// TIA Portal V18 export
// export: Created 2026-06-12T02:00:00Z, ExportSetting WithDefaults
VAR_GLOBAL   // PLC tag table "PLC_AI_B3_Tags"
   AI_B3_Sequence_Count AT %MD0 : Real;   // COUNT 0-100
   AI_B3_Flow_CIP_Center AT %MD4 : Real;   // FLOW 100-200 L/h
   AI_B3_Temp_CIP_Upper AT %MD8 : Real;   // TEMP 50-80 °C
   AI_B3_Pressure_CIP_1 AT %MD12 : Real;   // PRESSURE 7-8 bar
   AI_B3_Temp_Chaff_1 AT %MD16 : Real;   // TEMP 50-80 °C
   AI_B3_Flow_CIP_Feed AT %MD20 : Real;   // FLOW 100-200 L/h
   AI_B3_Temp_Steam_1 AT %MD24 : Real;   // TEMP 50-80 °C
   AI_B3_Flow_UCWW_1 AT %MD28 : Real;   // FLOW 100-200 L/h
   AI_B3_RPM_Screw_Conv AT %MD32 : Real;   // RPM 800-1200 RPM
   AI_B3_Temp_Condensate_1 AT %MD36 : Real;   // TEMP 50-80 °C
   AI_B3_Pressure_Screw_1 AT %MD40 : Real;   // PRESSURE 7-8 bar
   AI_B3_Flow_CWW_Out AT %MD44 : Real;   // FLOW 100-200 L/h
   AI_B3_Pressure_CWW_1 AT %MD48 : Real;   // PRESSURE 7-8 bar
   AI_B3_Temp_Decanter2 AT %MD52 : Real;   // TEMP 50-80 °C
   AI_B3_RPM_Rotary2 AT %MD56 : Real;   // RPM 800-1200 RPM
   AI_B3_RPM_Rotary1 AT %MD60 : Real;   // RPM 800-1200 RPM
   AI_B3_Temp_GroundSilo AT %MD64 : Real;   // TEMP 50-80 °C
   AI_B3_Flow_GroundSilo AT %MD68 : Real;   // FLOW 100-200 L/h
   AI_B3_Pressure_Mid_1 AT %MD72 : Real;   // PRESSURE 7-8 bar
   AI_B3_Flow_Condensate AT %MD76 : Real;   // FLOW 100-200 L/h
   AI_B3_Flow_Sump_Out AT %MD80 : Real;   // FLOW 100-200 L/h
   AI_B3_Level_Sump AT %MD84 : Real;   // LEVEL 30-80 %
   AI_B3_Pressure_Decant1 AT %MD88 : Real;   // PRESSURE 7-8 bar
   AI_B3_Pressure_Decant2 AT %MD92 : Real;   // PRESSURE 7-8 bar
   AI_B3_Flow_Decant1 AT %MD96 : Real;   // FLOW 100-200 L/h
   AI_B3_Temp_Decant1 AT %MD100 : Real;   // TEMP 50-80 °C
   AI_B3_Temp_FBB_Boiler AT %MD104 : Real;   // TEMP 50-80 °C
   AI_B3_Temp_CWW_Out AT %MD108 : Real;   // TEMP 50-80 °C
   AI_B3_Pressure_SUMP AT %MD112 : Real;   // PRESSURE 7-8 bar
   AI_B3_Flow_SUMP AT %MD116 : Real;   // FLOW 100-200 L/h
   AI_B3_Level_CWW AT %MD120 : Real;   // LEVEL 30-80 %
   AI_B3_Temp_FBB_Out AT %MD124 : Real;   // TEMP 50-80 °C
   AI_B3_Pressure_FBB_Out AT %MD128 : Real;   // PRESSURE 7-8 bar
   AI_B3_Flow_FBB_Out AT %MD132 : Real;   // FLOW 100-200 L/h
END_VAR
